// SIMATIC S7-200 SMART project (STEP 7-Micro/WIN SMART), CPU SR20

SYMBOL_TABLE System Symbols
Always_On        SM0.0    // Always ON
Clock_1s         SM0.5    // Clock pulse that is ON for 0.5 s, OFF for 0.5 s, for a duty cycle time of 1 s.
END_SYMBOL_TABLE

ORGANIZATION_BLOCK MAIN:OB1
TITLE=Program Comments
BEGIN
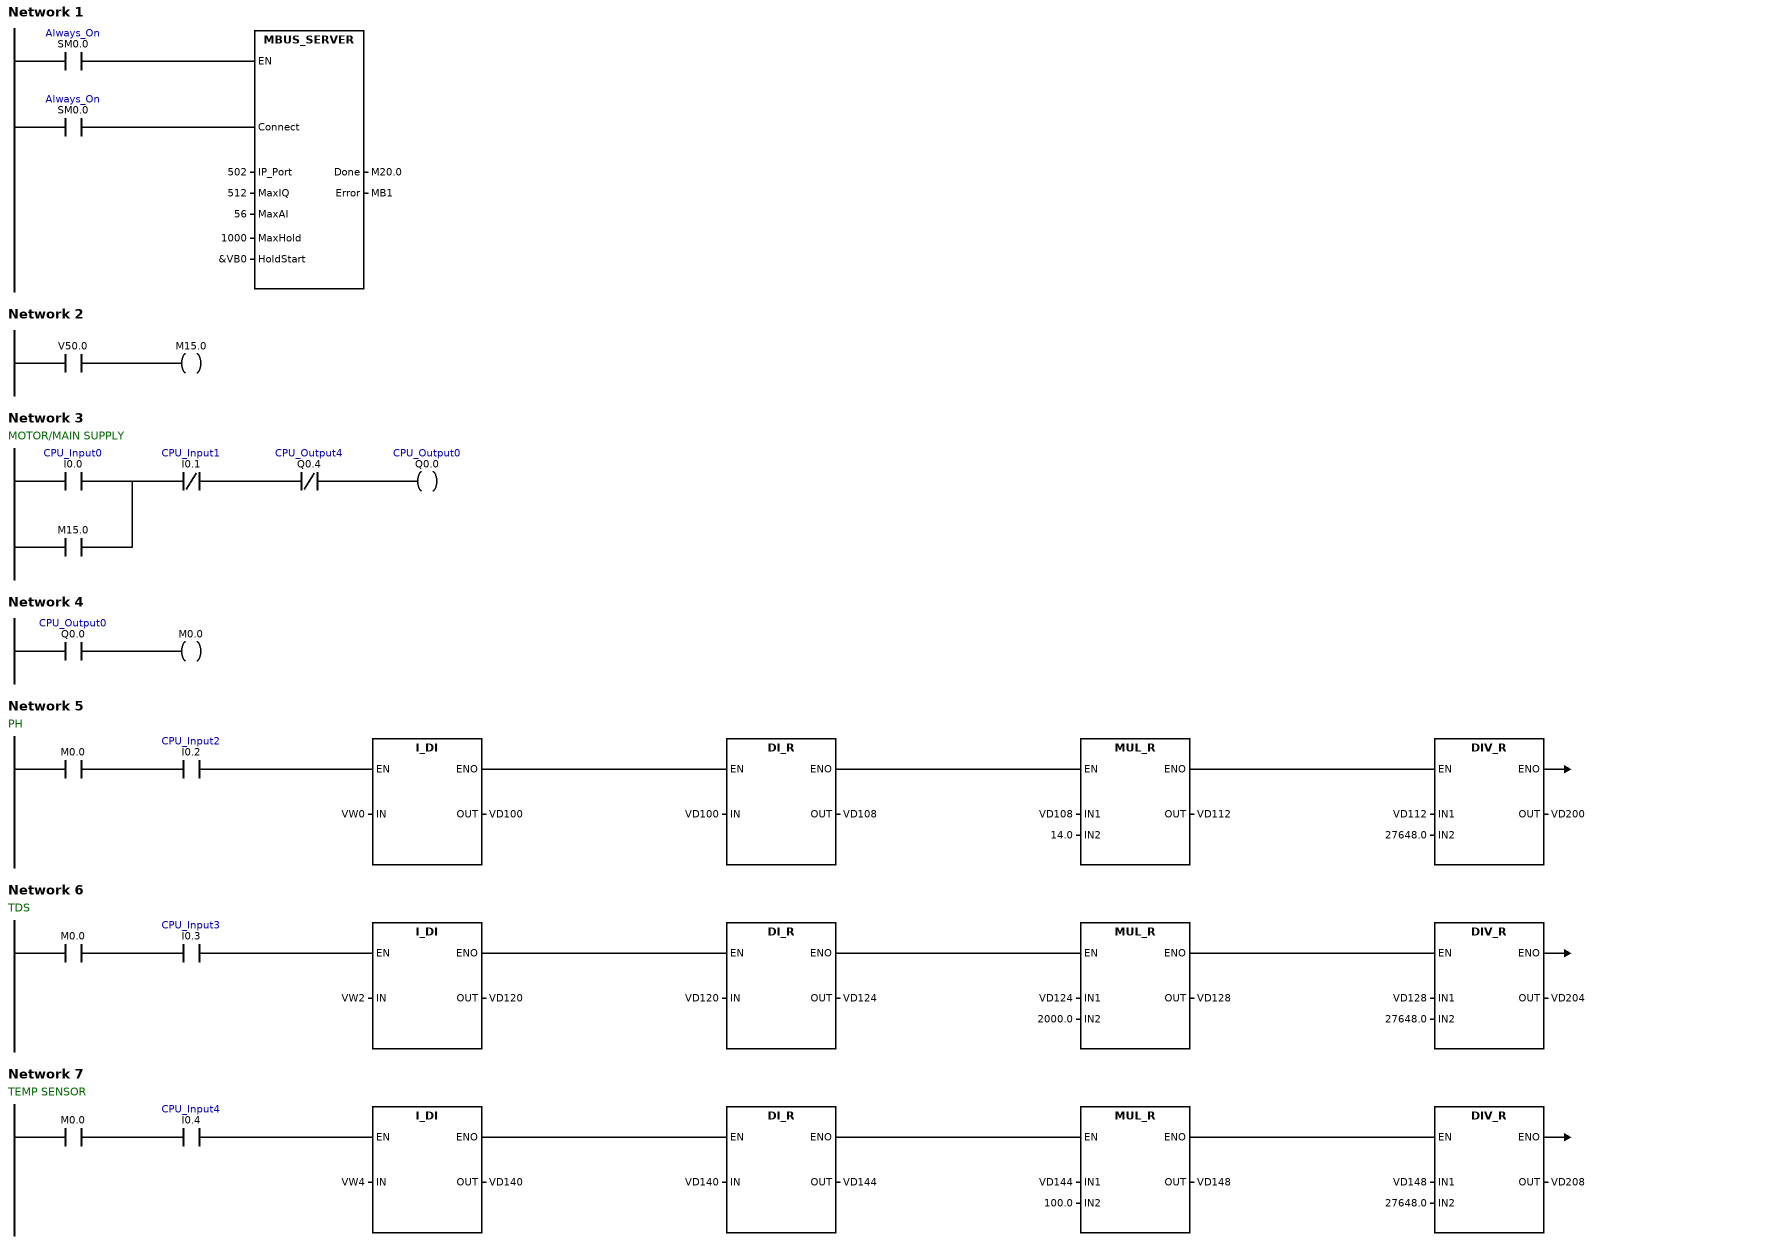
Network 1
LD     Always_On:SM0.0
=      L60.0
LD     Always_On:SM0.0
=      L63.7
LD     L60.0
CALL   MBUS_SERVER:SBR1, L63.7, 502, 512, 56, 1000, &VB0, M20.0, MB1
Network 2
LD     V50.0
=      M15.0
Network 3
// MOTOR/MAIN SUPPLY
LD     CPU_Input0:I0.0
O      M15.0
AN     CPU_Input1:I0.1
AN     CPU_Output4:Q0.4
=      CPU_Output0:Q0.0
Network 4
LD     CPU_Output0:Q0.0
=      M0.0
Network 5
// PH
LD     M0.0
A      CPU_Input2:I0.2
ITD    VW0, VD100
AENO
DTR    VD100, VD108
AENO
MOVR   VD108, VD112
AENO
*R     14.0, VD112
AENO
MOVR   VD112, VD200
/R     27648.0, VD200
Network 6
// TDS
LD     M0.0
A      CPU_Input3:I0.3
ITD    VW2, VD120
AENO
DTR    VD120, VD124
AENO
MOVR   VD124, VD128
AENO
*R     2000.0, VD128
AENO
MOVR   VD128, VD204
/R     27648.0, VD204
Network 7
// TEMP SENSOR
LD     M0.0
A      CPU_Input4:I0.4
ITD    VW4, VD140
AENO
DTR    VD140, VD144
AENO
MOVR   VD144, VD148
AENO
*R     100.0, VD148
AENO
MOVR   VD148, VD208
/R     27648.0, VD208
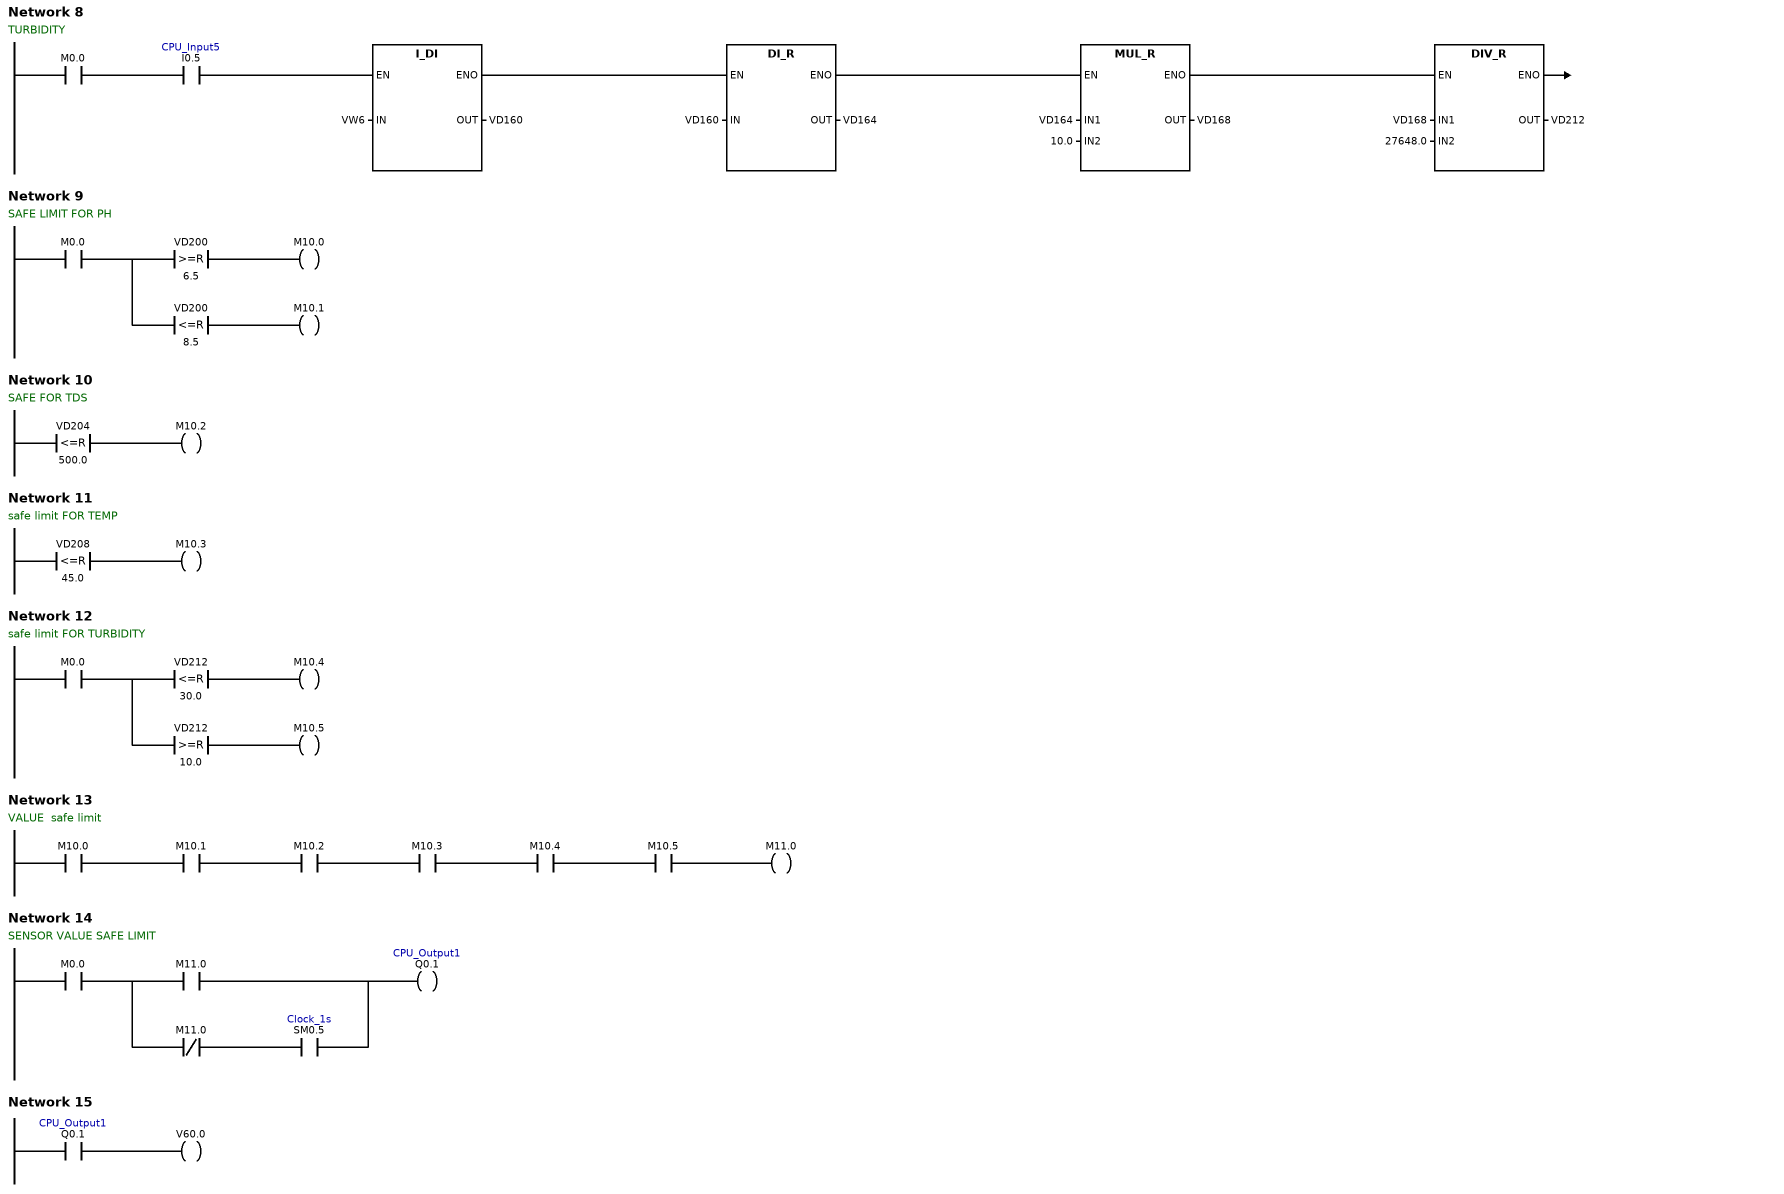
Network 8
// TURBIDITY
LD     M0.0
A      CPU_Input5:I0.5
ITD    VW6, VD160
AENO
DTR    VD160, VD164
AENO
MOVR   VD164, VD168
AENO
*R     10.0, VD168
AENO
MOVR   VD168, VD212
/R     27648.0, VD212
Network 9
// SAFE LIMIT FOR PH
LD     M0.0
LPS
AR>=   VD200, 6.5
=      M10.0
LPP
AR<=   VD200, 8.5
=      M10.1
Network 10
// SAFE FOR TDS
LDR<=  VD204, 500.0
=      M10.2
Network 11
//  safe limit FOR TEMP
LDR<=  VD208, 45.0
=      M10.3
Network 12
//  safe limit FOR TURBIDITY
LD     M0.0
LPS
AR<=   VD212, 30.0
=      M10.4
LPP
AR>=   VD212, 10.0
=      M10.5
Network 13
// VALUE  safe limit
LD     M10.0
A      M10.1
A      M10.2
A      M10.3
A      M10.4
A      M10.5
=      M11.0
Network 14
// SENSOR VALUE SAFE LIMIT
LD     M0.0
LD     M11.0
LDN    M11.0
A      Clock_1s:SM0.5
OLD
ALD
=      CPU_Output1:Q0.1
Network 15
LD     CPU_Output1:Q0.1
=      V60.0
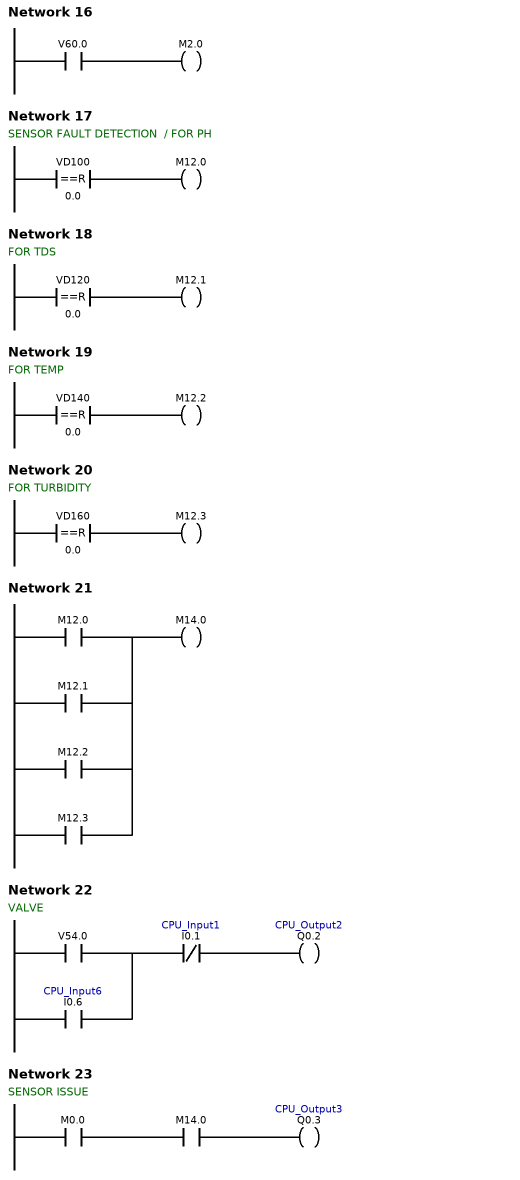
Network 16
LD     V60.0
=      M2.0
Network 17
// SENSOR FAULT DETECTION 
// FOR PH
LDR=   VD100, 0.0
=      M12.0
Network 18
// FOR TDS
LDR=   VD120, 0.0
=      M12.1
Network 19
// FOR TEMP
LDR=   VD140, 0.0
=      M12.2
Network 20
// FOR TURBIDITY
LDR=   VD160, 0.0
=      M12.3
Network 21
LD     M12.0
O      M12.1
O      M12.2
O      M12.3
=      M14.0
Network 22
// VALVE
// (network saved uncompiled; LAD cells follow)
// row 0: c0 -| |- V54.0 v  c1 -|/|- CPU_Input1:I0.1  c2 -( ) CPU_Output2:Q0.2
// row 1: c0 -| |- CPU_Input6:I0.6 ^
Network 23
// SENSOR ISSUE
LD     M0.0
A      M14.0
=      CPU_Output3:Q0.3
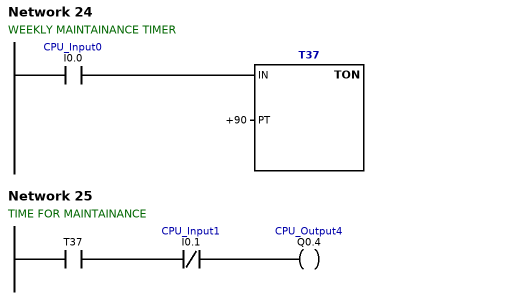
Network 24
// WEEKLY MAINTAINANCE TIMER
LD     CPU_Input0:I0.0
TON    T37, +90
Network 25
// TIME FOR MAINTAINANCE
LD     T37
AN     CPU_Input1:I0.1
=      CPU_Output4:Q0.4
END_ORGANIZATION_BLOCK

// SBR1: protected block, not included
